(* IEC 61131-3 sources: s22-soft-shell/st_interpret/tests/test_inputs/st_subset_3-4, 5 files *)

(* ---- 03_add.st ---- *)
PROGRAM 03_Add
VAR
    a: int;
END_VAR
a := (1 + 2);
END_PROGRAM

(* ---- 03_sub.st ---- *)
PROGRAM 03_Sub
VAR
    a: int;
END_VAR
a := (2 - 1);
END_PROGRAM

(* ---- 04_div.st ---- *)
PROGRAM 04_div
VAR
    a: int;
END_VAR
a := (10 / 2);
END_PROGRAM

(* ---- 04_mul.st ---- *)
PROGRAM 04_mul
VAR
    a: int;
END_VAR
a := (3 * 2);
END_PROGRAM

(* ---- 04_testA.st ---- *)
PROGRAM 04_testA
VAR
    a: int;
END_VAR
a := (2 + 4) * (1 + 3);
END_PROGRAM
